TYPE ST_WaferTransferParam :
STRUCT
	MaterialContext : ST_MaterialContext;
	Signal : ST_TransferHandshakeSignal;
END_STRUCT
END_TYPE

(* stored: Version 1.1.0.1, ProductVersion 3.1.4026.18
   DUT ST_WaferTransferParam: Id {8b20b1b5-25a3-4c7e-9f7a-c7836bf3a0a6} *)
